DATA_BLOCK "OUTPUTS DB"    DB60
TITLE =Shared digital outputs (multiple 410 subsystems)
// v0.1 - NEW tracked source, reconciled from two of Michou's uploads:
//   the raw "DB60 Outputs" export (2026-10-01, all fields still
//   Output_NNN placeholders) and his "FC155" rebuild upload (2026-10-02,
//   which already references two of these bits by new symbol names) -
//   the newer upload wins where they disagree, since it reflects a more
//   recent online edit:
//   - DBX7.6 (was Output_061) -> Calibration_Relay_K1... renamed
//     KILOTECK_Calib_K1 to match exactly what Michou's own FC155 upload
//     already references. K1 "Calibration Relay" - part of the KWS
//     CY300 power-up-defect workaround, see FC156.
//   - DBX7.7 (was Output_062) -> KILOTECK_Power_K2, same reasoning. K2
//     "Power Sw relay".
//   This IS the same "OUTPUTS DB" FC155 already references for
//   GRN_LED/RED_LED/WHT_SWL_1/2/3 (previously undocumented/untracked in
//   this repo as its own file) - confirmed by counting bit offsets in
//   the raw export: GRN_LED lands at DBX7.0, consistent with Michou's
//   literal "DB60.DBX7.6/DBX7.7" wording for K1/K2.
//   Flagged, not adopted here: Michou's FC155 upload also references
//   "OUTPUTS DB".WHT_SWL_1_Pnl/WHT_SWL_2_Pnl/WHT_SWL_3_Pnl/RED_LED_Pnl/
//   GRN_LED_Pnl (a "_Pnl" suffix) - the raw DB60 export used here still
//   has the plain names (WHT_SWL_1, RED_LED, GRN_LED, no suffix) that
//   FC155's own canonical source (this repo) already compiles against.
//   Kept the plain names since that's the only confirmed-current form;
//   if "_Pnl" is a real pending rename, re-export DB60 and this file
//   (and FC155's lamp/alarm networks) need updating together.
//   Every other field below (Output_NNN placeholders, Water_Valve,
//   Seam_Ctrl_*, tower lamps, etc.) is carried forward verbatim from
//   the raw export - not this subsystem's concern, not touched.
VERSION : 0.1


  STRUCT
   Output_0 : BOOL ;	//Temporary placeholder variable
   Output_01 : BOOL ;	//Temporary placeholder variable
   Output_02 : BOOL ;	//Temporary placeholder variable
   Output_03 : BOOL ;	//Temporary placeholder variable
   Output_04 : BOOL ;	//Temporary placeholder variable
   Output_05 : BOOL ;	//Temporary placeholder variable
   Output_06 : BOOL ;	//Temporary placeholder variable
   Output_07 : BOOL ;	//Temporary placeholder variable
   Water_Valve : BOOL ;	//Hot Water Valve  -> +N50
   Output_09 : BOOL ;	//Temporary placeholder variable
   Output_10 : BOOL ;
   Output_011 : BOOL ;	//Temporary placeholder variable
   Output_012 : BOOL ;	//Temporary placeholder variable
   Output_013 : BOOL ;	//Temporary placeholder variable
   Output_014 : BOOL ;	//Temporary placeholder variable
   Output_015 : BOOL ;	//Temporary placeholder variable
   Blu_Lamp : BOOL ;	//  -> +N50
   Red_Lamp : BOOL ;	//  -> +N50
   Buzzer_Out_A_B : BOOL ;	//  -> +N50
   Buzzer_Out_A_C : BOOL ;	//  -> +N50
   Buzzer_Out_ON : BOOL ;	//  -> +N50
   TuberStart_Disable : BOOL ;	//  -> +E07R
   Output_021 : BOOL ;	//Temporary placeholder variable
   Output_022 : BOOL ;	//Temporary placeholder variable
   Output_023 : BOOL ;	//Temporary placeholder variable
   Output_024 : BOOL ;	//Temporary placeholder variable
   Output_025 : BOOL ;	//Temporary placeholder variable
   Output_026 : BOOL ;	//Temporary placeholder variable
   BLUE_TOWERLAMP : BOOL ;	//- Q  3.4 Tower Light - Blu
   GREEN_TOWERLAMP : BOOL ;	//- Q  3.5 Tower Light - Grn
   RED_TOWERLAMP : BOOL ;	//- Q  3.5 Tower Light - Red
   ORANGE_TOWERLAMP : BOOL ;	//- Q  3.5 Tower Light - Org
   Output_031 : BOOL ;	//Temporary placeholder variable
   Output_032 : BOOL ;	//Temporary placeholder variable
   Output_033 : BOOL ;	//Temporary placeholder variable
   Output_034 : BOOL ;	//Temporary placeholder variable
   Output_035 : BOOL ;	//Temporary placeholder variable
   Output_036 : BOOL ;	//Temporary placeholder variable
   Output_037 : BOOL ;	//Temporary placeholder variable
   Output_038 : BOOL ;	//Temporary placeholder variable
   Seam_Ctrl_Power : BOOL ;	//-> +N75 ET200B (ADD5) Seam Ctrl B+ Relay
   Seam_Ctrl_Select : BOOL ;	//-> +N75 ET200B (ADD5) Seam Ctrl Select A/B  Relay
   Seam_Ctrl_Grn_SW_Lamp : BOOL ;	//-> +N75 ET200B (ADD5) GRN SW Lamp
   Seam_Ctrl_Wht_SW_Lamp : BOOL ;	//-> +N75 ET200B (ADD5) WHT SW Lamp
   Seam_Ctrl_Red_Top_Lamp : BOOL ;	//-> +N75 ET200B (ADD5) RED TOP Lamp
   Seam_Ctrl_Blu_Top_Lamp : BOOL ;	//-> +N75 ET200B (ADD5) BLU TOP Lamp
   Seam_Ctrl_Grn_Top_Lamp : BOOL ;	//-> +N75 ET200B (ADD5) GRN TOP Lamp
   Seam_Ctrl_Spare : BOOL ;	//-> +N75 ET200B (ADD5) Spare
   Output_047 : BOOL ;	//Temporary placeholder variable
   Output_048 : BOOL ;	//Temporary placeholder variable
   Output_049 : BOOL ;	//Temporary placeholder variable
   Output_050 : BOOL ;	//Temporary placeholder variable
   Output_051 : BOOL ;	//Temporary placeholder variable
   Output_052 : BOOL ;	//Temporary placeholder variable
   Output_053 : BOOL ;	//Temporary placeholder variable
   Output_054 : BOOL ;	//Temporary placeholder variable
   GRN_LED : BOOL ;	// - IO 8Bit Output ET-200B 8/8
   RED_LED : BOOL ;	// - IO 8Bit Output ET-200B 8/8
   WHT_SWL_1 : BOOL ;	// - IO 8Bit Output ET-200B 8/8
   WHT_SWL_2 : BOOL ;	// - IO 8Bit Output ET-200B 8/8
   WHT_SWL_3 : BOOL ;	// - IO 8Bit Output ET-200B 8/8
   Output_060 : BOOL ;	// - IO 8Bit Output ET-200B 8/8
   KILOTECK_Calib_K1 : BOOL ;	//DBX7.6 - K1 coil, PLC terminal 40 - applies the KWS CY300 shunt-cal loop, see FC156 (was Output_061)
   KILOTECK_Power_K2 : BOOL ;	//DBX7.7 - K2 coil, PLC terminal 39 - bridges KWS CY300 ON/OFF to Com, remote power pulse, see FC156 (was Output_062)
   Output_063 : BOOL ;	//Temporary placeholder variable
   Output_064 : BOOL ;	//Temporary placeholder variable
   Output_065 : BOOL ;	//Temporary placeholder variable
   Output_066 : BOOL ;	//Temporary placeholder variable
   Output_067 : BOOL ;	//Temporary placeholder variable
   Output_068 : BOOL ;	//Temporary placeholder variable
   Output_069 : BOOL ;	//Temporary placeholder variable
   Output_070 : BOOL ;	//Temporary placeholder variable
   Output_071 : BOOL ;	//Temporary placeholder variable
   Output_072 : BOOL ;	//Temporary placeholder variable
   Output_073 : BOOL ;	//Temporary placeholder variable
   Output_074 : BOOL ;	//Temporary placeholder variable
   Output_075 : BOOL ;	//Temporary placeholder variable
   Output_076 : BOOL ;	//Temporary placeholder variable
   Output_077 : BOOL ;	//Temporary placeholder variable
   Output_078 : BOOL ;	//Temporary placeholder variable
   Output_079 : BOOL ;	//Temporary placeholder variable
   Output_080 : BOOL ;	//Temporary placeholder variable
   Output_081 : BOOL ;	//Temporary placeholder variable
   Output_082 : BOOL ;	//Temporary placeholder variable
   Output_083 : BOOL ;	//Temporary placeholder variable
   Output_084 : BOOL ;	//Temporary placeholder variable
   Output_085 : BOOL ;	//Temporary placeholder variable
   Output_086 : BOOL ;	//Temporary placeholder variable
   Output_087 : BOOL ;	//Temporary placeholder variable
   Output_088 : BOOL ;	//Temporary placeholder variable
   Output_089 : BOOL ;	//Temporary placeholder variable
   Output_090 : BOOL ;	//Temporary placeholder variable
   Output_091 : BOOL ;	//Temporary placeholder variable
   Output_092 : BOOL ;	//Temporary placeholder variable
   Output_093 : BOOL ;	//Temporary placeholder variable
   Output_094 : BOOL ;	//Temporary placeholder variable
   Output_095 : BOOL ;	//Temporary placeholder variable
   Output_096 : BOOL ;	//Temporary placeholder variable
   Output_097 : BOOL ;	//Temporary placeholder variable
   Output_098 : BOOL ;	//Temporary placeholder variable
   Output_099 : BOOL ;	//Temporary placeholder variable
   Output_0100 : BOOL ;	//Temporary placeholder variable
   Output_0101 : BOOL ;	//Temporary placeholder variable
   Output_0102 : BOOL ;	//Temporary placeholder variable
   Output_0103 : BOOL ;	//Temporary placeholder variable
   Output_0104 : BOOL ;	//Temporary placeholder variable
   Output_0105 : BOOL ;	//Temporary placeholder variable
   Output_0106 : BOOL ;	//Temporary placeholder variable
   Output_0107 : BOOL ;	//Temporary placeholder variable
   Output_0108 : BOOL ;	//Temporary placeholder variable
   Output_0109 : BOOL ;	//Temporary placeholder variable
   Output_0110 : BOOL ;	//Temporary placeholder variable
   Output_0111 : BOOL ;	//Temporary placeholder variable
   Output_0112 : BOOL ;	//Temporary placeholder variable
   Output_0113 : BOOL ;	//Temporary placeholder variable
   Output_0114 : BOOL ;	//Temporary placeholder variable
   Output_0115 : BOOL ;	//Temporary placeholder variable
   Output_0116 : BOOL ;	//Temporary placeholder variable
   Output_0117 : BOOL ;	//Temporary placeholder variable
   Output_0118 : BOOL ;	//Temporary placeholder variable
   Output_0119 : BOOL ;	//Temporary placeholder variable
   Output_0120 : BOOL ;	//Temporary placeholder variable
   Output_0121 : BOOL ;	//Temporary placeholder variable
   Output_0122 : BOOL ;	//Temporary placeholder variable
   Output_0123 : BOOL ;	//Temporary placeholder variable
   Output_0124 : BOOL ;	//Temporary placeholder variable
   Output_0125 : BOOL ;	//Temporary placeholder variable
   Output_0126 : BOOL ;	//Temporary placeholder variable
   Output_0127 : BOOL ;	//Temporary placeholder variable
   Output_0128 : BOOL ;	//Temporary placeholder variable
   Output_0129 : BOOL ;	//Temporary placeholder variable
   Output_0130 : BOOL ;	//Temporary placeholder variable
   Output_0131 : BOOL ;	//Temporary placeholder variable
   Output_0132 : BOOL ;	//Temporary placeholder variable
   Output_0133 : BOOL ;	//Temporary placeholder variable
   Output_0134 : BOOL ;	//Temporary placeholder variable
   Output_0135 : BOOL ;	//Temporary placeholder variable
   Output_0136 : BOOL ;	//Temporary placeholder variable
   Output_0137 : BOOL ;	//Temporary placeholder variable
   Output_0138 : BOOL ;	//Temporary placeholder variable
   Output_0139 : BOOL ;	//Temporary placeholder variable
   Output_0140 : BOOL ;	//Temporary placeholder variable
   Output_0141 : BOOL ;	//Temporary placeholder variable
   Output_0142 : BOOL ;	//Temporary placeholder variable
   Output_0143 : BOOL ;	//Temporary placeholder variable
   Output_0144 : BOOL ;	//Temporary placeholder variable
   Output_0145 : BOOL ;	//Temporary placeholder variable
   Output_0146 : BOOL ;	//Temporary placeholder variable
   Output_0147 : BOOL ;	//Temporary placeholder variable
   Output_0148 : BOOL ;	//Temporary placeholder variable
   Output_0149 : BOOL ;	//Temporary placeholder variable
   Output_0150 : BOOL ;	//Temporary placeholder variable
   Output_0151 : BOOL ;	//Temporary placeholder variable
   Output_0152 : BOOL ;	//Temporary placeholder variable
   Output_0153 : BOOL ;	//Temporary placeholder variable
   Output_0154 : BOOL ;	//Temporary placeholder variable
   Output_0155 : BOOL ;	//Temporary placeholder variable
   Output_0156 : BOOL ;	//Temporary placeholder variable
   Output_0157 : BOOL ;	//Temporary placeholder variable
   Output_0158 : BOOL ;	//Temporary placeholder variable
   Output_0159 : BOOL ;	//Temporary placeholder variable
   Output_0160 : BOOL ;	//Temporary placeholder variable
   Output_0161 : BOOL ;	//Temporary placeholder variable
   Output_0162 : BOOL ;	//Temporary placeholder variable
   Output_0163 : BOOL ;	//Temporary placeholder variable
   Output_0164 : BOOL ;	//Temporary placeholder variable
   Output_0165 : BOOL ;	//Temporary placeholder variable
   Output_0166 : BOOL ;	//Temporary placeholder variable
   Output_0167 : BOOL ;	//Temporary placeholder variable
   Output_0168 : BOOL ;	//Temporary placeholder variable
   Output_0169 : BOOL ;	//Temporary placeholder variable
   Output_0170 : BOOL ;	//Temporary placeholder variable
   Output_0171 : BOOL ;	//Temporary placeholder variable
   Output_0172 : BOOL ;	//Temporary placeholder variable
   Output_0173 : BOOL ;	//Temporary placeholder variable
   Output_0174 : BOOL ;	//Temporary placeholder variable
   Output_0175 : BOOL ;	//Temporary placeholder variable
   Output_0176 : BOOL ;	//Temporary placeholder variable
   Output_0177 : BOOL ;	//Temporary placeholder variable
   Output_0178 : BOOL ;	//Temporary placeholder variable
   Output_0179 : BOOL ;	//Temporary placeholder variable
   Output_0180 : BOOL ;	//Temporary placeholder variable
   Output_0181 : BOOL ;	//Temporary placeholder variable
   Output_0182 : BOOL ;	//Temporary placeholder variable
   Output_0183 : BOOL ;	//Temporary placeholder variable
   Output_0184 : BOOL ;	//Temporary placeholder variable
   Output_0185 : BOOL ;	//Temporary placeholder variable
   Output_0186 : BOOL ;	//Temporary placeholder variable
   Output_0187 : BOOL ;	//Temporary placeholder variable
   Output_0188 : BOOL ;	//Temporary placeholder variable
   Output_0189 : BOOL ;	//Temporary placeholder variable
   Output_0190 : BOOL ;	//Temporary placeholder variable
   Output_0191 : BOOL ;	//Temporary placeholder variable
   Output_0192 : BOOL ;	//Temporary placeholder variable
   Output_0193 : BOOL ;	//Temporary placeholder variable
   Output_0194 : BOOL ;	//Temporary placeholder variable
   Output_0195 : BOOL ;	//Temporary placeholder variable
   Output_0196 : BOOL ;	//Temporary placeholder variable
   Output_0197 : BOOL ;	//Temporary placeholder variable
   Output_0198 : BOOL ;	//Temporary placeholder variable
   Output_0199 : BOOL ;	//Temporary placeholder variable
   Output_0200 : BOOL ;	//Temporary placeholder variable
   Output_0201 : BOOL ;	//Temporary placeholder variable
   Output_0202 : BOOL ;	//Temporary placeholder variable
   Output_0203 : BOOL ;	//Temporary placeholder variable
   Output_0204 : BOOL ;	//Temporary placeholder variable
   Output_0205 : BOOL ;	//Temporary placeholder variable
   Output_0206 : BOOL ;	//Temporary placeholder variable
   Output_0207 : BOOL ;	//Temporary placeholder variable
   Output_0208 : BOOL ;	//Temporary placeholder variable
   Output_0209 : BOOL ;	//Temporary placeholder variable
   Output_0210 : BOOL ;	//Temporary placeholder variable
   Output_0211 : BOOL ;	//Temporary placeholder variable
   Output_0212 : BOOL ;	//Temporary placeholder variable
   Output_0213 : BOOL ;	//Temporary placeholder variable
   Output_0214 : BOOL ;	//Temporary placeholder variable
   Output_0215 : BOOL ;	//Temporary placeholder variable
   Output_0216 : BOOL ;	//Temporary placeholder variable
   Output_0217 : BOOL ;	//Temporary placeholder variable
   Output_0218 : BOOL ;	//Temporary placeholder variable
   Output_0219 : BOOL ;	//Temporary placeholder variable
   Output_0220 : BOOL ;	//Temporary placeholder variable
   Output_0221 : BOOL ;	//Temporary placeholder variable
   Output_0222 : BOOL ;	//Temporary placeholder variable
   Output_0223 : BOOL ;	//Temporary placeholder variable
   Output_0224 : BOOL ;	//Temporary placeholder variable
   Output_0225 : BOOL ;	//Temporary placeholder variable
   Output_0226 : BOOL ;	//Temporary placeholder variable
   Output_0227 : BOOL ;	//Temporary placeholder variable
   Output_0228 : BOOL ;	//Temporary placeholder variable
   Output_0229 : BOOL ;	//Temporary placeholder variable
   Output_0230 : BOOL ;	//Temporary placeholder variable
   Output_0231 : BOOL ;	//Temporary placeholder variable
   Output_0232 : BOOL ;	//Temporary placeholder variable
   Output_0233 : BOOL ;	//Temporary placeholder variable
   Output_0234 : BOOL ;	//Temporary placeholder variable
   Output_0235 : BOOL ;	//Temporary placeholder variable
   Output_0236 : BOOL ;	//Temporary placeholder variable
   Output_0237 : BOOL ;	//Temporary placeholder variable
   Output_0238 : BOOL ;	//Temporary placeholder variable
   Output_0239 : BOOL ;	//Temporary placeholder variable
   Output_0240 : BOOL ;	//Temporary placeholder variable
   Output_0241 : BOOL ;	//Temporary placeholder variable
   Output_0242 : BOOL ;	//Temporary placeholder variable
   Output_0243 : BOOL ;	//Temporary placeholder variable
   Output_0244 : BOOL ;	//Temporary placeholder variable
   Output_0245 : BOOL ;	//Temporary placeholder variable
   Output_0246 : BOOL ;	//Temporary placeholder variable
   Output_0247 : BOOL ;	//Temporary placeholder variable
   Output_0248 : BOOL ;	//Temporary placeholder variable
   Output_0249 : BOOL ;	//Temporary placeholder variable
   Output_0250 : BOOL ;	//Temporary placeholder variable
   Output_0251 : BOOL ;	//Temporary placeholder variable
   Output_0252 : BOOL ;	//Temporary placeholder variable
   Output_0253 : BOOL ;	//Temporary placeholder variable
   Output_0254 : BOOL ;	//Temporary placeholder variable
   Output_0255 : BOOL ;	//Temporary placeholder variable
   Output_0256 : BOOL ;	//Temporary placeholder variable
   Output_0257 : BOOL ;	//Temporary placeholder variable
   Output_0258 : BOOL ;	//Temporary placeholder variable
   Output_0259 : BOOL ;	//Temporary placeholder variable
   Output_0260 : BOOL ;	//Temporary placeholder variable
   Output_0261 : BOOL ;	//Temporary placeholder variable
   Output_0262 : BOOL ;	//Temporary placeholder variable
   Output_0263 : BOOL ;	//Temporary placeholder variable
   Output_0264 : BOOL ;	//Temporary placeholder variable
   Output_0265 : BOOL ;	//Temporary placeholder variable
   Output_0266 : BOOL ;	//Temporary placeholder variable
   Output_0267 : BOOL ;	//Temporary placeholder variable
   Output_0268 : BOOL ;	//Temporary placeholder variable
   Output_0269 : BOOL ;	//Temporary placeholder variable
   Output_0270 : BOOL ;	//Temporary placeholder variable
   Output_0271 : BOOL ;	//Temporary placeholder variable
  END_STRUCT ;
BEGIN
   Output_0 := FALSE;
   Output_01 := FALSE;
   Output_02 := FALSE;
   Output_03 := FALSE;
   Output_04 := FALSE;
   Output_05 := FALSE;
   Output_06 := FALSE;
   Output_07 := FALSE;
   Water_Valve := FALSE;
   Output_09 := FALSE;
   Output_10 := FALSE;
   Output_011 := FALSE;
   Output_012 := FALSE;
   Output_013 := FALSE;
   Output_014 := FALSE;
   Output_015 := FALSE;
   Blu_Lamp := FALSE;
   Red_Lamp := FALSE;
   Buzzer_Out_A_B := FALSE;
   Buzzer_Out_A_C := FALSE;
   Buzzer_Out_ON := FALSE;
   TuberStart_Disable := FALSE;
   Output_021 := FALSE;
   Output_022 := FALSE;
   Output_023 := FALSE;
   Output_024 := FALSE;
   Output_025 := FALSE;
   Output_026 := FALSE;
   BLUE_TOWERLAMP := FALSE;
   GREEN_TOWERLAMP := FALSE;
   RED_TOWERLAMP := FALSE;
   ORANGE_TOWERLAMP := FALSE;
   Output_031 := FALSE;
   Output_032 := FALSE;
   Output_033 := FALSE;
   Output_034 := FALSE;
   Output_035 := FALSE;
   Output_036 := FALSE;
   Output_037 := FALSE;
   Output_038 := FALSE;
   Seam_Ctrl_Power := FALSE;
   Seam_Ctrl_Select := FALSE;
   Seam_Ctrl_Grn_SW_Lamp := FALSE;
   Seam_Ctrl_Wht_SW_Lamp := FALSE;
   Seam_Ctrl_Red_Top_Lamp := FALSE;
   Seam_Ctrl_Blu_Top_Lamp := FALSE;
   Seam_Ctrl_Grn_Top_Lamp := FALSE;
   Seam_Ctrl_Spare := FALSE;
   Output_047 := FALSE;
   Output_048 := FALSE;
   Output_049 := FALSE;
   Output_050 := FALSE;
   Output_051 := FALSE;
   Output_052 := FALSE;
   Output_053 := FALSE;
   Output_054 := FALSE;
   GRN_LED := FALSE;
   RED_LED := FALSE;
   WHT_SWL_1 := FALSE;
   WHT_SWL_2 := FALSE;
   WHT_SWL_3 := FALSE;
   Output_060 := FALSE;
   KILOTECK_Calib_K1 := FALSE;
   KILOTECK_Power_K2 := FALSE;
   Output_063 := FALSE;
   Output_064 := FALSE;
   Output_065 := FALSE;
   Output_066 := FALSE;
   Output_067 := FALSE;
   Output_068 := FALSE;
   Output_069 := FALSE;
   Output_070 := FALSE;
   Output_071 := FALSE;
   Output_072 := FALSE;
   Output_073 := FALSE;
   Output_074 := FALSE;
   Output_075 := FALSE;
   Output_076 := FALSE;
   Output_077 := FALSE;
   Output_078 := FALSE;
   Output_079 := FALSE;
   Output_080 := FALSE;
   Output_081 := FALSE;
   Output_082 := FALSE;
   Output_083 := FALSE;
   Output_084 := FALSE;
   Output_085 := FALSE;
   Output_086 := FALSE;
   Output_087 := FALSE;
   Output_088 := FALSE;
   Output_089 := FALSE;
   Output_090 := FALSE;
   Output_091 := FALSE;
   Output_092 := FALSE;
   Output_093 := FALSE;
   Output_094 := FALSE;
   Output_095 := FALSE;
   Output_096 := FALSE;
   Output_097 := FALSE;
   Output_098 := FALSE;
   Output_099 := FALSE;
   Output_0100 := FALSE;
   Output_0101 := FALSE;
   Output_0102 := FALSE;
   Output_0103 := FALSE;
   Output_0104 := FALSE;
   Output_0105 := FALSE;
   Output_0106 := FALSE;
   Output_0107 := FALSE;
   Output_0108 := FALSE;
   Output_0109 := FALSE;
   Output_0110 := FALSE;
   Output_0111 := FALSE;
   Output_0112 := FALSE;
   Output_0113 := FALSE;
   Output_0114 := FALSE;
   Output_0115 := FALSE;
   Output_0116 := FALSE;
   Output_0117 := FALSE;
   Output_0118 := FALSE;
   Output_0119 := FALSE;
   Output_0120 := FALSE;
   Output_0121 := FALSE;
   Output_0122 := FALSE;
   Output_0123 := FALSE;
   Output_0124 := FALSE;
   Output_0125 := FALSE;
   Output_0126 := FALSE;
   Output_0127 := FALSE;
   Output_0128 := FALSE;
   Output_0129 := FALSE;
   Output_0130 := FALSE;
   Output_0131 := FALSE;
   Output_0132 := FALSE;
   Output_0133 := FALSE;
   Output_0134 := FALSE;
   Output_0135 := FALSE;
   Output_0136 := FALSE;
   Output_0137 := FALSE;
   Output_0138 := FALSE;
   Output_0139 := FALSE;
   Output_0140 := FALSE;
   Output_0141 := FALSE;
   Output_0142 := FALSE;
   Output_0143 := FALSE;
   Output_0144 := FALSE;
   Output_0145 := FALSE;
   Output_0146 := FALSE;
   Output_0147 := FALSE;
   Output_0148 := FALSE;
   Output_0149 := FALSE;
   Output_0150 := FALSE;
   Output_0151 := FALSE;
   Output_0152 := FALSE;
   Output_0153 := FALSE;
   Output_0154 := FALSE;
   Output_0155 := FALSE;
   Output_0156 := FALSE;
   Output_0157 := FALSE;
   Output_0158 := FALSE;
   Output_0159 := FALSE;
   Output_0160 := FALSE;
   Output_0161 := FALSE;
   Output_0162 := FALSE;
   Output_0163 := FALSE;
   Output_0164 := FALSE;
   Output_0165 := FALSE;
   Output_0166 := FALSE;
   Output_0167 := FALSE;
   Output_0168 := FALSE;
   Output_0169 := FALSE;
   Output_0170 := FALSE;
   Output_0171 := FALSE;
   Output_0172 := FALSE;
   Output_0173 := FALSE;
   Output_0174 := FALSE;
   Output_0175 := FALSE;
   Output_0176 := FALSE;
   Output_0177 := FALSE;
   Output_0178 := FALSE;
   Output_0179 := FALSE;
   Output_0180 := FALSE;
   Output_0181 := FALSE;
   Output_0182 := FALSE;
   Output_0183 := FALSE;
   Output_0184 := FALSE;
   Output_0185 := FALSE;
   Output_0186 := FALSE;
   Output_0187 := FALSE;
   Output_0188 := FALSE;
   Output_0189 := FALSE;
   Output_0190 := FALSE;
   Output_0191 := FALSE;
   Output_0192 := FALSE;
   Output_0193 := FALSE;
   Output_0194 := FALSE;
   Output_0195 := FALSE;
   Output_0196 := FALSE;
   Output_0197 := FALSE;
   Output_0198 := FALSE;
   Output_0199 := FALSE;
   Output_0200 := FALSE;
   Output_0201 := FALSE;
   Output_0202 := FALSE;
   Output_0203 := FALSE;
   Output_0204 := FALSE;
   Output_0205 := FALSE;
   Output_0206 := FALSE;
   Output_0207 := FALSE;
   Output_0208 := FALSE;
   Output_0209 := FALSE;
   Output_0210 := FALSE;
   Output_0211 := FALSE;
   Output_0212 := FALSE;
   Output_0213 := FALSE;
   Output_0214 := FALSE;
   Output_0215 := FALSE;
   Output_0216 := FALSE;
   Output_0217 := FALSE;
   Output_0218 := FALSE;
   Output_0219 := FALSE;
   Output_0220 := FALSE;
   Output_0221 := FALSE;
   Output_0222 := FALSE;
   Output_0223 := FALSE;
   Output_0224 := FALSE;
   Output_0225 := FALSE;
   Output_0226 := FALSE;
   Output_0227 := FALSE;
   Output_0228 := FALSE;
   Output_0229 := FALSE;
   Output_0230 := FALSE;
   Output_0231 := FALSE;
   Output_0232 := FALSE;
   Output_0233 := FALSE;
   Output_0234 := FALSE;
   Output_0235 := FALSE;
   Output_0236 := FALSE;
   Output_0237 := FALSE;
   Output_0238 := FALSE;
   Output_0239 := FALSE;
   Output_0240 := FALSE;
   Output_0241 := FALSE;
   Output_0242 := FALSE;
   Output_0243 := FALSE;
   Output_0244 := FALSE;
   Output_0245 := FALSE;
   Output_0246 := FALSE;
   Output_0247 := FALSE;
   Output_0248 := FALSE;
   Output_0249 := FALSE;
   Output_0250 := FALSE;
   Output_0251 := FALSE;
   Output_0252 := FALSE;
   Output_0253 := FALSE;
   Output_0254 := FALSE;
   Output_0255 := FALSE;
   Output_0256 := FALSE;
   Output_0257 := FALSE;
   Output_0258 := FALSE;
   Output_0259 := FALSE;
   Output_0260 := FALSE;
   Output_0261 := FALSE;
   Output_0262 := FALSE;
   Output_0263 := FALSE;
   Output_0264 := FALSE;
   Output_0265 := FALSE;
   Output_0266 := FALSE;
   Output_0267 := FALSE;
   Output_0268 := FALSE;
   Output_0269 := FALSE;
   Output_0270 := FALSE;
   Output_0271 := FALSE;
END_DATA_BLOCK

